# B&R Automation Studio project Test-repository
Automation Studio 4.5.2.102

## Configuration Config1

CPU 4PPC70.0702-20B, AutomationRuntime D4.52, Build 4.1.2, Vc V4.52.0

### Task classes (Cpu.sw)
```
Cyclic#4:
  LoveLD <- LoveLD.prg
VcDataObjects: Visu <- Visu.dob
```

### Hardware
```
4PPC70_0702_20B : 4PPC70.0702-20B v1.4.0.0
  Connector IF2:
    ActivateDevice = 1
  VcObjectName = Visu
  KeyMappingFile = VC\4PPC70_0702_20B.dis
```

## Logical view

### Global.typ - Global data types
```iecst
TYPE
	di_type : 	STRUCT  (*digital inputs*)
		PressureSwitch : BOOL;
	END_STRUCT;
	do_type : 	STRUCT  (*digital outputs*)
		RedStackLight : BOOL;
	END_STRUCT;
END_TYPE
```

### Global.var - Global variables
```iecst
VAR
	gdo : do_type; (*process variable for do type*)
	gExecute : BOOL;
	gdi : di_type; (*process variable for di type*)
END_VAR
```

- Visualisation Logical/Visu (not shown)

### Program Logical/LoveLD (IEC)

#### Cyclic.ld
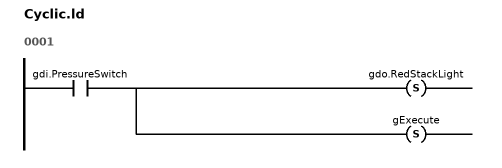
Ladder, written as Structured Text:
```iecst
PROGRAM _CYCLIC
(* Network 1 *)
IF gdi.PressureSwitch THEN
    gdo.RedStackLight := TRUE;
    gExecute := TRUE;
END_IF;
END_PROGRAM
```

### Program Logical/NewProgram

#### Variables.var
```iecst
VAR
	Start : BOOL;
	Begin : INT;
END_VAR
```

#### Main.st
```iecst
PROGRAM _INIT
	(* Insert code here *)

END_PROGRAM

PROGRAM _CYCLIC

	IF Start THEN
		Begin := 1;
	END_IF

END_PROGRAM

PROGRAM _EXIT
	(* Insert code here *)

END_PROGRAM
```

Listed in the project but not available here: Logical/Libraries
